(* CODESYS project WagoLibWeatherUnderground_v0.0.1.library
   Company: WAGO Corp. USA
   Title: WagoLibWeatherunderground
   Description: This library contains function blocks to get weather from Weather Underground web service.
   Author: Jesse Cox
   Version: 0.0.1

Project tree, tasks and I/O mapping:
  libraries: ; WagoSysString, * (WAGO); SysProcess, 3.5.7.0 (System); SysTypes2 Interfaces, 3.5.4.0 (System); WagoAppFileDir, 1.6.1.1 (WAGO)
  function block fbWeatherUnderGround [ST]: CurlCurrentWeather
  data type WEATHER
*)

// WEATHER
TYPE WEATHER :
STRUCT
	sWeatherString		: STRING;
	rTempF				: REAL;
	rTempC				: REAL;
	rRelativeHumidity	: REAL;
	sWindString			: STRING;
	sWindDirection		: STRING;
	rWindDegrees		: REAL;
	rWindSpeedMph		: REAL;
	rWindGustMph		: REAL;
	rWindSpeedKph		: REAL;
	rWindGustKph		: REAL;
	rPressureMb			: REAL;
	rPressureIn			: REAL;
	rDewpointF			: REAL;
	rDewpointC			: REAL;
	rWindchillF			: REAL;
	rWindchillC			: REAL;
	rFeelslikeF			: REAL;
	rFeelslikeC			: REAL;
	rVisibilityMi		: REAL;
	rVisibilityKm		: REAL; 
	rPrecipitationIn	: REAL;
END_STRUCT
END_TYPE

// fbWeatherUnderGround
FUNCTION_BLOCK fbWeatherUnderGround
VAR_IN_OUT
	xExecute			: BOOL;
END_VAR
VAR_INPUT
	sApiKey				: STRING;
	sState				: STRING;
	sCity				: STRING;
END_VAR
VAR_OUTPUT
	typLocalWeather		: WEATHER;
END_VAR
VAR
	fbReadFile: FbReadWholeFile_cpt;
	oReadFileStatus: FbResult;
	xReadFileTrigger: BOOL;
	xReadFileError: BOOL;
	xReadFileBusy: BOOL;
	sReadFileName: STRING := '/root/weather.json';
	aReadFileData: ARRAY[0..10000] OF BYTE;
	iReadFileSize: UDINT := 3000;
	iReadFileNumOfBytes: UDINT;
	xReadFileEndOfFileReached: BOOL;
	i: UDINT;
	
	sStringInProcess	: STRING;
	sProcessedStrings	: ARRAY[0..200] OF STRING;
	xIsCharacter: BOOL;
	ftCurlDoneTrig	: F_TRIG;
	rtFileIsDone	: R_TRIG;
	rtNotCharacter	: R_TRIG;
	iCharCount: INT;
END_VAR

IF xExecute THEN
	CurlCurrentWeather(sApiKey:= sApiKey, sApiState:= sState, sApiCity:= sCity);
	xReadFileTrigger := TRUE;
END_IF

fbReadFile(
	oStatus=> oReadFileStatus, 
	xTrigger:= xReadFileTrigger, 
	xError=> xReadFileError, 
	xBusy=> xReadFileBusy, 
	sName:= sReadFileName, 
	pRxBuffer:= ADR(aReadFileData), 
	udiRxBufferSize:= iReadFileSize, 
	udiRxNBytes=> iReadFileNumOfBytes, 
	xEofReached=> xReadFileEndOfFileReached);
	
rtFileIsDone(CLK:= xReadFileEndOfFileReached);
iCharCount := 0; // reset the string count for processing
IF rtFileIsDone.Q THEN	
	FOR i := 0 TO iReadFileNumOfBytes DO
		IF 	((aReadFileData[i] >= 48) AND (aReadFileData[i] <= 57)) OR // characters 0-9
			((aReadFileData[i] >= 65) AND (aReadFileData[i] <= 90)) OR // characters A-Z
			((aReadFileData[i] >= 97) AND (aReadFileData[i] <= 122)) THEN // characters a-z
				xIsCharacter := TRUE;
		ELSIF 	(aReadFileData[i] = 34) OR // character "
				(aReadFileData[i] = 44) OR // character ,
				(aReadFileData[i] = 123) OR // character {
				(aReadFileData[i] = 125) THEN // character }
					xIsCharacter := FALSE;
		END_IF
	
		IF xIsCharacter THEN
			sStringInProcess := CONCAT(sStringInProcess, ASCIIBYTE_TO_STRING(aReadFileData[i]));
			sProcessedStrings[iCharCount] := sStringInProcess;
		END_IF
			
		rtNotCharacter(CLK := NOT xIsCharacter);
		IF rtNotCharacter.Q THEN
			sStringInProcess := '';
			iCharCount := iCharCount + 1;
		END_IF
	END_FOR
	FOR i := 0 TO iCharCount DO
		IF sProcessedStrings[i] = 'weather' THEN
			typLocalWeather.sWeatherString := sProcessedStrings[i + 1];	
		ELSIF sProcessedStrings[i] = 'temp_f' THEN
			typLocalWeather.rTempF := STRING_TO_REAL(sProcessedStrings[i + 1]);
		ELSIF sProcessedStrings[i] = 'temp_c' THEN
			typLocalWeather.rTempC := STRING_TO_REAL(sProcessedStrings[i + 1]);
		ELSIF sProcessedStrings[i] = 'relative_humidity' THEN
			typLocalWeather.rRelativeHumidity := STRING_TO_REAL(sProcessedStrings[i + 1]);
		ELSIF sProcessedStrings[i] = 'wind_string' THEN
			typLocalWeather.sWindString := sProcessedStrings[i + 1];
		ELSIF sProcessedStrings[i] = 'wind_dir' THEN
			typLocalWeather.sWindDirection := sProcessedStrings[i + 1];
		ELSIF sProcessedStrings[i] = 'wind_degrees' THEN
			typLocalWeather.rWindDegrees := STRING_TO_REAL(sProcessedStrings[i + 1]);
		ELSIF sProcessedStrings[i] = 'wind_mph' THEN
			typLocalWeather.rWindSpeedMph := STRING_TO_REAL(sProcessedStrings[i + 1]);
		ELSIF sProcessedStrings[i] = 'wind_gust_mph' THEN
			typLocalWeather.rWindGustMph := STRING_TO_REAL(sProcessedStrings[i + 1]);
		ELSIF sProcessedStrings[i] = 'wind_kph' THEN
			typLocalWeather.rWindSpeedKph := STRING_TO_REAL(sProcessedStrings[i + 1]);
		ELSIF sProcessedStrings[i] = 'wind_gust_kph' THEN
			typLocalWeather.rWindGustKph := STRING_TO_REAL(sProcessedStrings[i + 1]);
		ELSIF sProcessedStrings[i] = 'pressure_mb' THEN
			typLocalWeather.rPressureMb := STRING_TO_REAL(sProcessedStrings[i + 1]);
		ELSIF sProcessedStrings[i] = 'pressure_in' THEN
			typLocalWeather.rPressureIn := STRING_TO_REAL(sProcessedStrings[i + 1]);
		ELSIF sProcessedStrings[i] = 'dewpoint_f' THEN
			typLocalWeather.rDewpointF := STRING_TO_REAL(sProcessedStrings[i + 1]);
		ELSIF sProcessedStrings[i] = 'dewpoint_c' THEN
			typLocalWeather.rDewpointC := STRING_TO_REAL(sProcessedStrings[i + 1]);
		ELSIF sProcessedStrings[i] = 'windchill_f' THEN
			typLocalWeather.rWindchillF := STRING_TO_REAL(sProcessedStrings[i + 1]);
		ELSIF sProcessedStrings[i] = 'windchill_c' THEN
			typLocalWeather.rWindchillC := STRING_TO_REAL(sProcessedStrings[i + 1]);
		ELSIF sProcessedStrings[i] = 'feelslike_f' THEN
			typLocalWeather.rFeelslikeF := STRING_TO_REAL(sProcessedStrings[i + 1]);
		ELSIF sProcessedStrings[i] = 'feelslike_c' THEN
			typLocalWeather.rFeelslikeC := STRING_TO_REAL(sProcessedStrings[i + 1]);
		ELSIF sProcessedStrings[i] = 'visibility_mi' THEN
			typLocalWeather.rVisibilityMi := STRING_TO_REAL(sProcessedStrings[i + 1]);
		ELSIF sProcessedStrings[i] = 'visibility_km' THEN
			typLocalWeather.rVisibilityKm:= STRING_TO_REAL(sProcessedStrings[i + 1]);
		ELSIF sProcessedStrings[i] = 'precip_today_in' THEN
			typLocalWeather.rPrecipitationIn:= STRING_TO_REAL(sProcessedStrings[i + 1]);
		END_IF
	END_FOR
	xExecute := FALSE;
END_IF

METHOD CurlCurrentWeather : STRING
VAR_INPUT
	sApiKey		: STRING;
	sApiState	: STRING;
	sApiCity	: STRING;
END_VAR
VAR 
	sUprString	: STRING(255);// := 'curl --insecure --output /root/weather.json -X GET http://api.wunderground.com/api/';	// base string to query weather service
	pRslt: POINTER TO RTS_IEC_RESULT;
	diCurl: DINT;
	diFileStatus: DINT;
	sQueryBashScript: STRING;
	sBashResponse: STRING;
	ptBashRslt: POINTER TO RTS_IEC_RESULT;
END_VAR
sUprString := 'curl --insecure --output /root/weather.json -X GET http://api.wunderground.com/api/';
sUprString := CONCAT(sUprString, sApiKey);
sUprString := CONCAT(sUprString, '/conditions/q/');
sUprString := CONCAT(sUprString, sApiState);
sUprString := CONCAT(sUprString, '/');
sUprString := CONCAT(sUprString, sApiCity);
sUprString := CONCAT(sUprString, '.json');

diFileStatus := SysProcessExecuteCommand2(pszCommand:= sUprString, pszStdOut:= sBashResponse, udiStdOutLen:= LEN(sUprString), pResult:= ptBashRslt);
//curl --insecure --output /root/weather.json -X GET http://api.wunderground.com/api/1ad24b0986c7e326/conditions/q/OR/Portland.json
END_METHOD

END_FUNCTION_BLOCK
